(* IEC 61131-3 sources: repolevel_ST_code_completion/output/0122完整版本_无planner目前sota/repoeval_plc_hello_mixing_tank/readful_result_no_provide, 6 files *)

(* ---- F_ResetDeviceCommands.st ---- *)
// 混合电机命令复位
	IF bMixerRunning THEN
		bMixerRunCmd := FALSE;		// 已运行，复位运行命令
	ELSE
		bMixerStopCmd := FALSE;		// 已停止，复位停止命令
	END_IF;

	// 介质1阀门命令复位
	IF bMedium1Opened THEN
		bMedium1OpenCmd := FALSE;	// 已打开，复位打开命令
	ELSE
		bMedium1CloseCmd := FALSE;	// 已关闭，复位关闭命令
	END_IF;

	// 介质2阀门命令复位
	IF bMedium2Opened THEN
		bMedium2OpenCmd := FALSE;	// 已打开，复位打开命令
	ELSE
		bMedium2CloseCmd := FALSE;	// 已关闭，复位关闭命令
	END_IF;

	// 排水阀门命令复位
	IF bDrainOpened THEN
		bDrainOpenCmd := FALSE;		// 已打开，复位打开命令
	ELSE
		bDrainCloseCmd := FALSE;	// 已关闭，复位关闭命令
	END_IF;

	RETURN;
END_FUNCTION

(* ---- F_UpdateLimitSwitches.st ---- *)
bLevelFull := rTankLevel >= rFullThreshold;		// 液位 >= 满阈值时，满开关激活
bLevelEmpty := rTankLevel <= rEmptyThreshold;	// 液位 <= 空阈值时，空开关激活

F_UpdateLimitSwitches := TRUE;
RETURN;
END_FUNCTION

(* ---- FB_AutoSequence.st ---- *)
VAR
	tonMixing			:	TON;			// 混合定时器
END_VAR

// 复位逻辑
IF bReset THEN
	eCurrentState := AUTO_SEQUENCE.DRAINING;
	nCyclesCompleted := 0;
END_IF

// 自动序列状态机
IF bEnable THEN
	CASE eCurrentState OF
		AUTO_SEQUENCE.FILLING:
			// 确保其他设备不工作
			bMixerRunCmd := FALSE;
			bDrainOpenCmd := FALSE;

			// 开启介质阀门
			bMedium1OpenCmd := TRUE;
			bMedium2OpenCmd := TRUE;

			// 检查液位满传感器
			IF bTankLevelFull THEN
				bMedium1OpenCmd := FALSE;
				bMedium2OpenCmd := FALSE;
				eCurrentState := AUTO_SEQUENCE.MIXING;
			END_IF;

		AUTO_SEQUENCE.MIXING:
			// 确保其他设备不工作
			bMedium1OpenCmd := FALSE;
			bMedium2OpenCmd := FALSE;
			bDrainOpenCmd := FALSE;

			// 开启混合电机
			bMixerRunCmd := TRUE;

			// 启动混合定时器
			tonMixing(IN := TRUE, PT := tMixingDuration);

			// 检查定时器是否完成
			IF tonMixing.Q THEN
				bMixerRunCmd := FALSE;
				eCurrentState := AUTO_SEQUENCE.DRAINING;
			END_IF;

		AUTO_SEQUENCE.DRAINING:
			// 确保其他设备不工作
			bMixerRunCmd := FALSE;
			bMedium1OpenCmd := FALSE;
			bMedium2OpenCmd := FALSE;

			// 开启排空阀门
			bDrainOpenCmd := TRUE;

			// 检查液位空传感器
			IF bTankLevelEmpty THEN
				bDrainOpenCmd := FALSE;
				eCurrentState := AUTO_SEQUENCE.FILLING;
				nCyclesCompleted := nCyclesCompleted + 1;
			END_IF;

		ELSE
			// 默认状态，确保所有设备关闭
			bMixerRunCmd := FALSE;
			bMedium1OpenCmd := FALSE;
			bMedium2OpenCmd := FALSE;
			bDrainOpenCmd := FALSE;
	END_CASE;
END_IF;
END_FUNCTION_BLOCK

(* ---- FB_ManualControl.st ---- *)
VAR
	bMedium1Latch		:	BOOL;
	bMedium2Latch		:	BOOL;
	bDrainLatch			:	BOOL;
END_VAR

// 混合电机控制
bMixerRunCmdOut := (bMixerRunCmd OR bMixerRunning) AND NOT bMixerStopCmd;

// 介质阀1控制
bMedium1Latch := (bMedium1OpenCmd OR bMedium1Opened) AND NOT bMedium1CloseCmd;
bMedium1OpenCmdOut := bMedium1Latch;

// 介质阀2控制
bMedium2Latch := (bMedium2OpenCmd OR bMedium2Opened) AND NOT bMedium2CloseCmd;
bMedium2OpenCmdOut := bMedium2Latch;

// 排放阀控制
bDrainLatch := (bDrainOpenCmd OR bDrainOpened) AND NOT bDrainCloseCmd;
bDrainOpenCmdOut := bDrainLatch;
END_FUNCTION_BLOCK

(* ---- FB_ModeController.st ---- *)
VAR
	eLastMode		:	MODES;	// 上次模式
END_VAR

// 模式切换逻辑
CASE eCurrentMode OF
	MODES.AUTO:
		IF bSetToManual THEN
			eCurrentMode := MODES.MANUAL;
		END_IF

	MODES.MANUAL:
		IF bSetToAuto THEN
			eCurrentMode := MODES.AUTO;
		END_IF
END_CASE

// 检测模式变化
bModeChanged := (eCurrentMode <> eLastMode);
eLastMode := eCurrentMode;
END_FUNCTION_BLOCK

(* ---- FB_TankLevelSimulator.st ---- *)
VAR
	rNewLevel : REAL; // 临时变量，用于计算新的液位
END_VAR

// 复位逻辑
IF bReset THEN
	rCurrentLevel := rInitialLevel;
ELSE
	// 液位计算
	rNewLevel := rCurrentLevel
				+ rFillRate1 * BOOL_TO_REAL(bMedium1Opened)
				+ rFillRate2 * BOOL_TO_REAL(bMedium2Opened)
				- rDrainRate * BOOL_TO_REAL(bDrainOpened);

	// 确保液位在最小和最大范围内
	IF rNewLevel < rMinLevel THEN
		rCurrentLevel := rMinLevel;
	ELSIF rNewLevel > rMaxLevel THEN
		rCurrentLevel := rMaxLevel;
	ELSE
		rCurrentLevel := rNewLevel;
	END_IF;
END_IF;
END_FUNCTION_BLOCK
